(* CODESYS project losowanie.project

Project tree, tasks and I/O mapping:
  Device : CODESYS Control Win V3, 3S - Smart Software Solutions GmbH, order no. 305021, version 3.5.8.10
    application Application
      libraries: Standard, * (System); VisuDialogs, * (System)
      task MainTask (cyclic, interval t#20ms, priority 1) calls PLC_PRG
      task VISU_TASK (cyclic, interval 100 ms, priority 31) calls VisuElems.Visu_Prg
      program PLC_PRG [ST]
      visualisation Visualization
  text list GlobalTextList
*)

// Device/Application/PLC_PRG
PROGRAM PLC_PRG
VAR
	_TIME: TON;
	COUNTER : CTU;
	DELAY : CTU;
	RAND_1: WORD;
	RAND_2: WORD;
	RAND_3: WORD;
	RAND_4: WORD;
	
	INPUT_1 : WORD;
	INPUT_2 : WORD;
	INPUT_3 : WORD;
	INPUT_4 : WORD;
	INPUT_5 : WORD;
	COME_IN : BOOL := TRUE;
	
	IS_OVER : WSTRING := "GRA TRWA";
END_VAR

_TIME(PT:=T#1MS, IN := NOT _TIME.Q);
COUNTER(CU:=_TIME.Q, RESET:=COUNTER.Q, PV:=71);

IF COUNTER.CV > 10 AND COUNTER.CV < 70 AND COME_IN THEN	
	RAND_1:=(ROR(SHR(COUNTER.CV, 1),COUNTER.CV MOD 7)MOD 9) +1;
	RAND_2:=((SHR(COUNTER.CV,2)*17) MOD 9) +1;
	RAND_3:=(ROR(SHR(COUNTER.CV, 2),COUNTER.CV MOD 7)MOD 9) +1;
	RAND_4:=((SHR(COUNTER.CV,2)*13) MOD 9) +1;
	IF RAND_1 <> RAND_2 THEN
		COME_IN := FALSE;
	END_IF
END_IF

IF	INPUT_1 <> 0 AND INPUT_2 <> 0 AND INPUT_3 <> 0 AND INPUT_4 <> 0 AND INPUT_5 <> 0 THEN
	IF (RAND_1 + RAND_4 + INPUT_2 = 9) AND (RAND_2 + INPUT_3 + INPUT_4 = 9) AND (INPUT_1 + INPUT_5 + RAND_3 = 9)
	AND (RAND_1 + RAND_2 + INPUT_1 = 9) AND (INPUT_2 + INPUT_3 + RAND_3 = 9) AND (RAND_4 + INPUT_4 + INPUT_5 = 9)
	THEN
		IS_OVER := "GRA ZAKOŃCZONA SUKCESEM";
	ELSE
		IS_OVER := "GRA ZAKOŃCZONA NIEPOWODZENIEM";
	END_IF
END_IF

END_PROGRAM

// Device/Application/Visualization
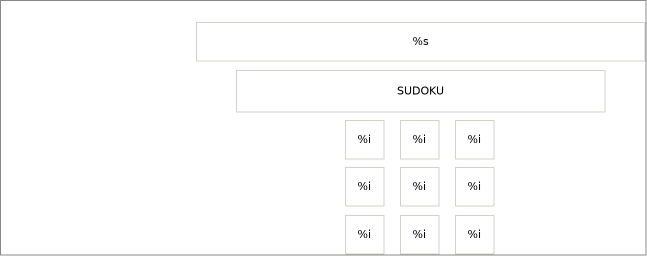
VISUALIZATION Visualization  // 647x256
    Textfield (345,120 39x39), "%i", text variable: PLC_PRG.RAND_1
    Textfield (345,167 39x39), "%i", text variable: PLC_PRG.RAND_2
    Textfield (345,215 39x39), "%i", text variable: PLC_PRG.INPUT_1
        OnMouseClick: write the text variable via VisuDialogs.Numpad
    Textfield (400,120 39x39), "%i", text variable: PLC_PRG.INPUT_2
        OnMouseClick: write the text variable via VisuDialogs.Numpad
    Textfield (400,167 39x39), "%i", text variable: PLC_PRG.INPUT_3
        OnMouseClick: write the text variable via VisuDialogs.Numpad
    Textfield (400,215 39x39), "%i", text variable: PLC_PRG.RAND_3
    Textfield (455,167 39x39), "%i", text variable: PLC_PRG.INPUT_4
        OnMouseClick: write the text variable via VisuDialogs.Numpad
    Textfield (455,215 39x39), "%i", text variable: PLC_PRG.INPUT_5
        OnMouseClick: write the text variable via VisuDialogs.Numpad
    Textfield (196,22 449x39), "%s", text variable: PLC_PRG.IS_OVER
    Textfield (455,120 39x39), "%i", text variable: PLC_PRG.RAND_4
    Textfield (236,70 369x42), "SUDOKU"
END_VISUALIZATION
